FUNCTION_BLOCK Sensor_Comunicacao_HMI (* Service Interface Function Block Type *)
  (* Standard: 61499-2 *)
  (* Version 0.0, 20/01/2026, Schneider Electric, template *)
  PACKAGE Hidryco.HidrycoLib;
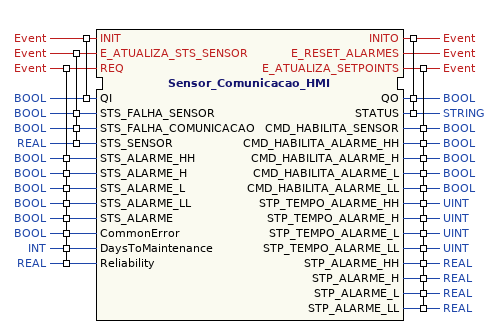
  EVENT_INPUT
    INIT WITH QI;
    E_ATUALIZA_STS_SENSOR WITH STS_SENSOR, STS_FALHA_SENSOR, STS_FALHA_COMUNICACAO;
    REQ WITH STS_ALARME_HH, STS_ALARME_H, STS_ALARME_L, STS_ALARME_LL, STS_ALARME, CommonError, DaysToMaintenance, Reliability;
  END_EVENT
  EVENT_OUTPUT
    INITO WITH QO, STATUS;
    E_RESET_ALARMES;
    E_ATUALIZA_SETPOINTS WITH STP_TEMPO_ALARME_HH, STP_TEMPO_ALARME_H, STP_TEMPO_ALARME_L, STP_TEMPO_ALARME_LL, STP_ALARME_HH, STP_ALARME_H, STP_ALARME_L, STP_ALARME_LL, CMD_HABILITA_SENSOR, CMD_HABILITA_ALARME_HH, CMD_HABILITA_ALARME_H, CMD_HABILITA_ALARME_L, CMD_HABILITA_ALARME_LL;
  END_EVENT
  VAR_INPUT
    QI : BOOL;
    STS_FALHA_SENSOR : BOOL;
    STS_FALHA_COMUNICACAO : BOOL;
    STS_SENSOR : REAL;
    STS_ALARME_HH : BOOL;
    STS_ALARME_H : BOOL;
    STS_ALARME_L : BOOL;
    STS_ALARME_LL : BOOL;
    STS_ALARME : BOOL;
    CommonError : BOOL;
    DaysToMaintenance : INT;
    Reliability : REAL;
  END_VAR
  VAR_OUTPUT
    QO : BOOL; (* Event Output Qualifier *)
    STATUS : STRING; (* Service Status *)
    CMD_HABILITA_SENSOR : BOOL;
    CMD_HABILITA_ALARME_HH : BOOL;
    CMD_HABILITA_ALARME_H : BOOL;
    CMD_HABILITA_ALARME_L : BOOL;
    CMD_HABILITA_ALARME_LL : BOOL;
    STP_TEMPO_ALARME_HH : UINT;
    STP_TEMPO_ALARME_H : UINT;
    STP_TEMPO_ALARME_L : UINT;
    STP_TEMPO_ALARME_LL : UINT;
    STP_ALARME_HH : REAL;
    STP_ALARME_H : REAL;
    STP_ALARME_L : REAL;
    STP_ALARME_LL : REAL;
  END_VAR
  SERVICE /
    SEQUENCE 
    END_SEQUENCE
  END_SERVICE
END_FUNCTION_BLOCK
